FUNCTION_BLOCK MainStation EXTENDS TcoCore.TcoObject
VAR
    turckRfidHead : RfidHead(THIS^, T#1MS);
    sUId : T_MaxString;
    _uid : BOOL;
END_VAR

turckRfidHead();

IF _uid THEN
    turckRfidHead.ReadUidMethod();
    _uid := FALSE;
END_IF

IF turckRfidHead.ReadUidTask.Done then
    sUId := turckRfidHead.sUId;
END_IF

END_FUNCTION_BLOCK

(* stored: Version 1.1.0.1, ProductVersion 3.1.4024.12
   POU MainStation: Id {e386d5e3-cce4-00c5-305e-24e2ac159f53}, SpecialFunc None *)
